(* Logix 5000 project; controller PLC vendor 1 type 14 code 155 rev 32.13; software revision 32.04; part 4 of 5 *)
(* tags used below, declared in another part *)
   Bridge_Timer_Gearing_Delay : TIMER;
   Bridge_Timer_Gearing_Delay_DN_OS : BOOL;
   Bridge_Timer_Gearing_Duration : TIMER;
   Bridge_Timer_Gearing_Duration_DN_OS : BOOL;
   Bypass_Encoder : BOOL;   // HMI ENABLE ENCODER
   Depositor : Depositor_R2b;
   Depositor_Bridge_Up : BOOL;
   Depositor_Spout_Done_OS : BOOL[32];
   Encoder_Conveyor : AXIS_CIP_DRIVE;
   IO : IO_R2a;
   MV_conveyor_stopped : BOOL;
   MV_Encoder_Stop_Value : REAL;
   mv_index_counter : COUNTER;
   NC_NF : NCNF_R2a;   // NC/NF BITSHIFTS
   OS : INT[10];
   Recipe_Setpoints_DINT : DINT[23,20];
   Release_Bridge_Distance : REAL[10];
   Release_MAG_Distance : REAL[10];
   Releases_Dive : BOOL;
   Sequencer_Auto : Sequencer_R2a;
   Sequencer_Home : Sequencer_R2a;
   Servo_Bridge_Shift : AXIS_CIP_DRIVE;
   Servo_MC_Bridge_Shift : Axis_MC_R3b;
   System : System_R2e;
   TEST_COUNTER : COUNTER;
   TEST_COUNTER_2 : COUNTER;
   Timers : TIMER[20];   // x
(* MainProgram, continued *)

ROUTINE File_100_Servo_Bridge   (* ladder *)
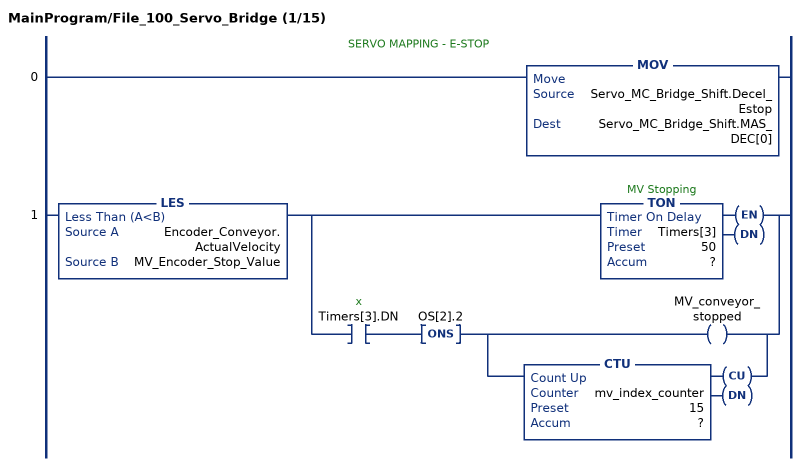
   // SERVO MAPPING - E-STOP
   0: MOV(Servo_MC_Bridge_Shift.Decel_Estop,Servo_MC_Bridge_Shift.MAS_DEC[0]);
   1: LES(Encoder_Conveyor.ActualVelocity,MV_Encoder_Stop_Value)[TON(Timers[3],?,?) ,XIC(Timers[3].DN) ONS(OS[2].2) [OTE(MV_conveyor_stopped) ,CTU(mv_index_counter,?,?) ] ];
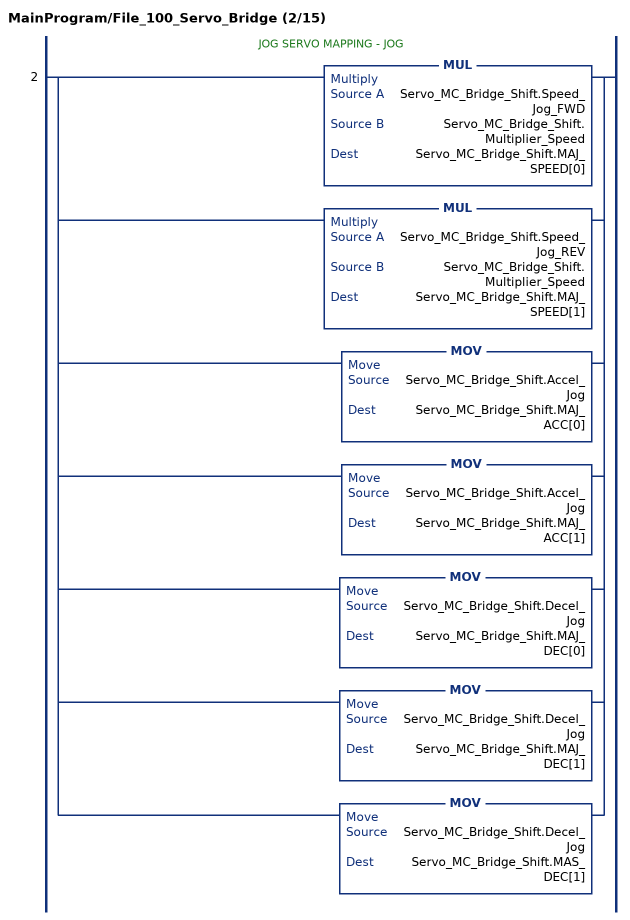
   // JOG SERVO MAPPING - JOG
   2: [MUL(Servo_MC_Bridge_Shift.Speed_Jog_FWD,Servo_MC_Bridge_Shift.Multiplier_Speed,Servo_MC_Bridge_Shift.MAJ_SPEED[0]) ,MUL(Servo_MC_Bridge_Shift.Speed_Jog_REV,Servo_MC_Bridge_Shift.Multiplier_Speed,Servo_MC_Bridge_Shift.MAJ_SPEED[1]) ,MOV(Servo_MC_Bridge_Shift.Accel_Jog,Servo_MC_Bridge_Shift.MAJ_ACC[0]) ,MOV(Servo_MC_Bridge_Shift.Accel_Jog,Servo_MC_Bridge_Shift.MAJ_ACC[1]) ,MOV(Servo_MC_Bridge_Shift.Decel_Jog,Servo_MC_Bridge_Shift.MAJ_DEC[0]) ,MOV(Servo_MC_Bridge_Shift.Decel_Jog,Servo_MC_Bridge_Shift.MAJ_DEC[1]) ,MOV(Servo_MC_Bridge_Shift.Decel_Jog,Servo_MC_Bridge_Shift.MAS_DEC[1]) ];
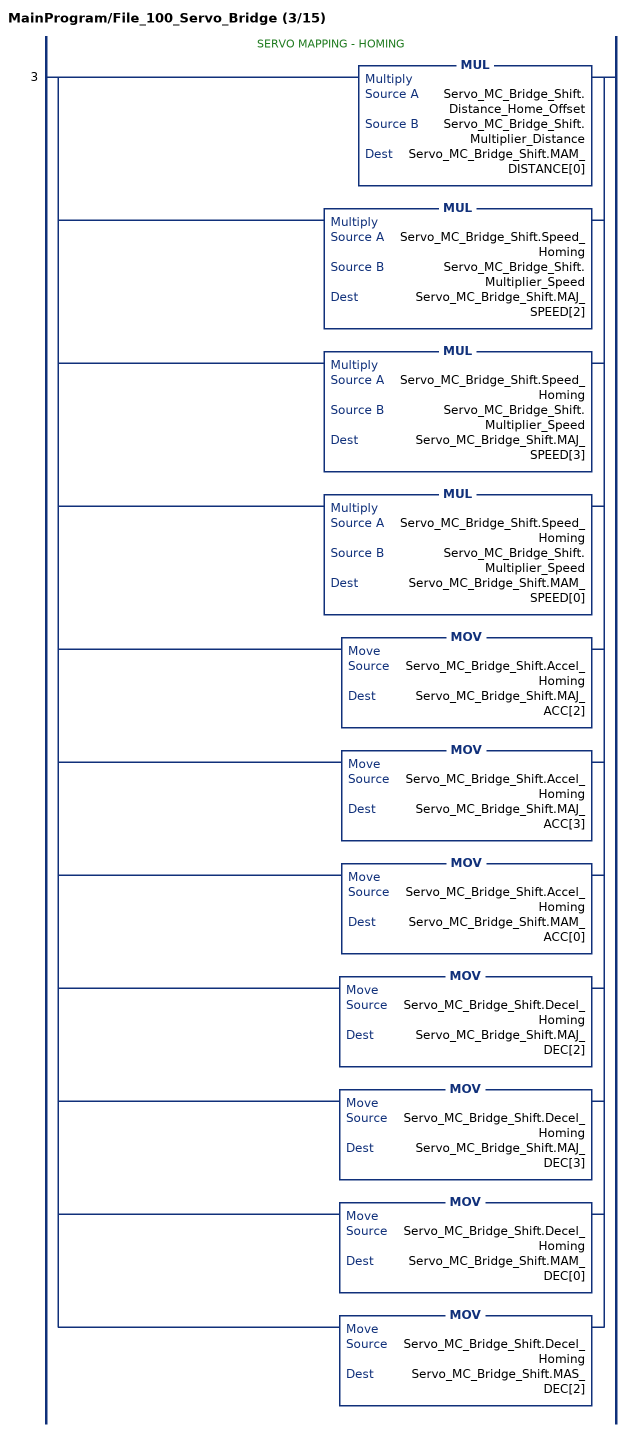
   // SERVO MAPPING - HOMING
   3: [MUL(Servo_MC_Bridge_Shift.Distance_Home_Offset,Servo_MC_Bridge_Shift.Multiplier_Distance,Servo_MC_Bridge_Shift.MAM_DISTANCE[0]) ,MUL(Servo_MC_Bridge_Shift.Speed_Homing,Servo_MC_Bridge_Shift.Multiplier_Speed,Servo_MC_Bridge_Shift.MAJ_SPEED[2]) ,MUL(Servo_MC_Bridge_Shift.Speed_Homing,Servo_MC_Bridge_Shift.Multiplier_Speed,Servo_MC_Bridge_Shift.MAJ_SPEED[3]) ,MUL(Servo_MC_Bridge_Shift.Speed_Homing,Servo_MC_Bridge_Shift.Multiplier_Speed,Servo_MC_Bridge_Shift.MAM_SPEED[0]) ,MOV(Servo_MC_Bridge_Shift.Accel_Homing,Servo_MC_Bridge_Shift.MAJ_ACC[2]) ,MOV(Servo_MC_Bridge_Shift.Accel_Homing,Servo_MC_Bridge_Shift.MAJ_ACC[3]) ,MOV(Servo_MC_Bridge_Shift.Accel_Homing,Servo_MC_Bridge_Shift.MAM_ACC[0]) ,MOV(Servo_MC_Bridge_Shift.Decel_Homing,Servo_MC_Bridge_Shift.MAJ_DEC[2]) ,MOV(Servo_MC_Bridge_Shift.Decel_Homing,Servo_MC_Bridge_Shift.MAJ_DEC[3]) ,MOV(Servo_MC_Bridge_Shift.Decel_Homing,Servo_MC_Bridge_Shift.MAM_DEC[0]) ,MOV(Servo_MC_Bridge_Shift.Decel_Homing,Servo_MC_Bridge_Shift.MAS_DEC[2]) ];
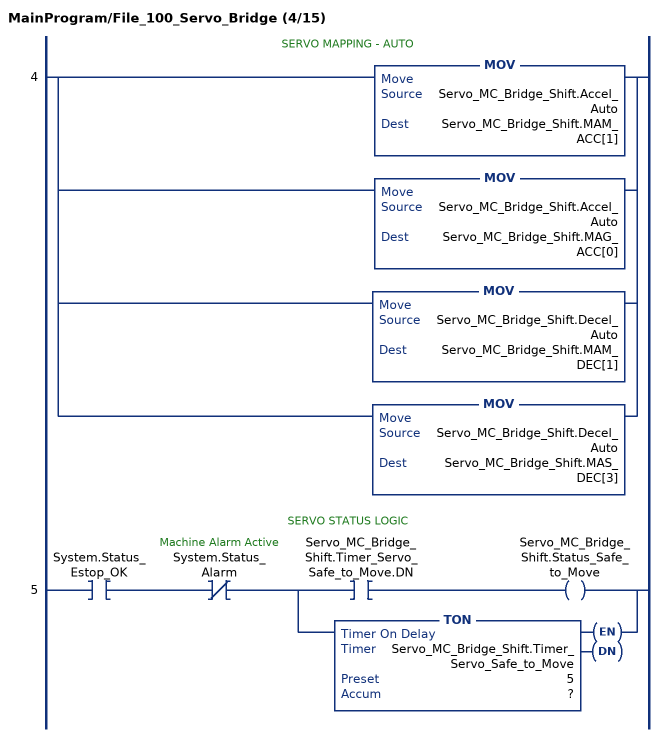
   // SERVO MAPPING - AUTO
   4: [MOV(Servo_MC_Bridge_Shift.Accel_Auto,Servo_MC_Bridge_Shift.MAM_ACC[1]) ,MOV(Servo_MC_Bridge_Shift.Accel_Auto,Servo_MC_Bridge_Shift.MAG_ACC[0]) ,MOV(Servo_MC_Bridge_Shift.Decel_Auto,Servo_MC_Bridge_Shift.MAM_DEC[1]) ,MOV(Servo_MC_Bridge_Shift.Decel_Auto,Servo_MC_Bridge_Shift.MAS_DEC[3]) ];
   // SERVO STATUS LOGIC
   5: XIC(System.Status_Estop_OK)XIO(System.Status_Alarm)[XIC(Servo_MC_Bridge_Shift.Timer_Servo_Safe_to_Move.DN) OTE(Servo_MC_Bridge_Shift.Status_Safe_to_Move) ,TON(Servo_MC_Bridge_Shift.Timer_Servo_Safe_to_Move,?,?) ];
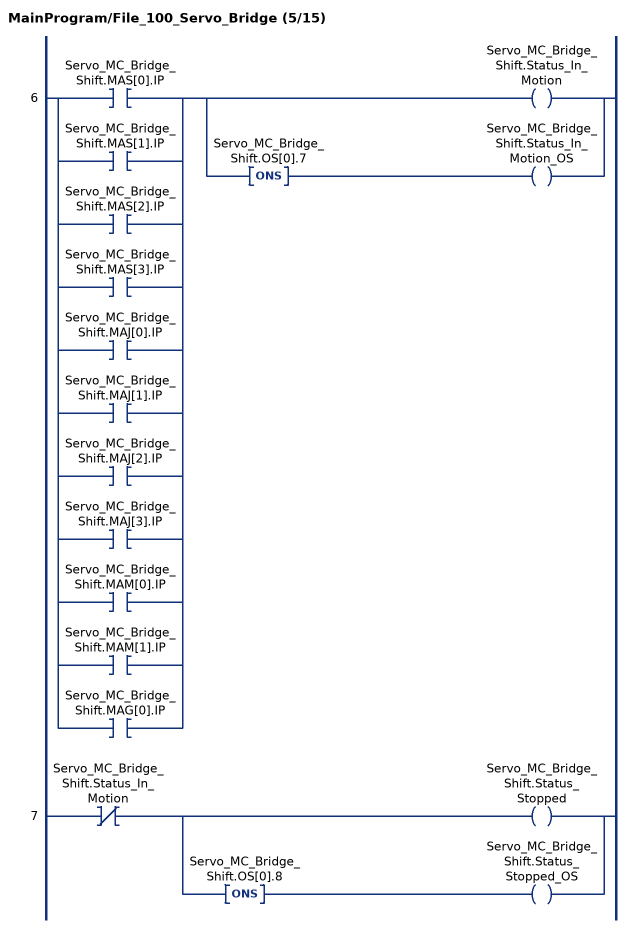
   6: [XIC(Servo_MC_Bridge_Shift.MAS[0].IP) ,XIC(Servo_MC_Bridge_Shift.MAS[1].IP) ,XIC(Servo_MC_Bridge_Shift.MAS[2].IP) ,XIC(Servo_MC_Bridge_Shift.MAS[3].IP) ,XIC(Servo_MC_Bridge_Shift.MAJ[0].IP) ,XIC(Servo_MC_Bridge_Shift.MAJ[1].IP) ,XIC(Servo_MC_Bridge_Shift.MAJ[2].IP) ,XIC(Servo_MC_Bridge_Shift.MAJ[3].IP) ,XIC(Servo_MC_Bridge_Shift.MAM[0].IP) ,XIC(Servo_MC_Bridge_Shift.MAM[1].IP) ,XIC(Servo_MC_Bridge_Shift.MAG[0].IP) ][OTE(Servo_MC_Bridge_Shift.Status_In_Motion) ,ONS(Servo_MC_Bridge_Shift.OS[0].7) OTE(Servo_MC_Bridge_Shift.Status_In_Motion_OS) ];
   7: XIO(Servo_MC_Bridge_Shift.Status_In_Motion)[OTE(Servo_MC_Bridge_Shift.Status_Stopped) ,ONS(Servo_MC_Bridge_Shift.OS[0].8) OTE(Servo_MC_Bridge_Shift.Status_Stopped_OS) ];
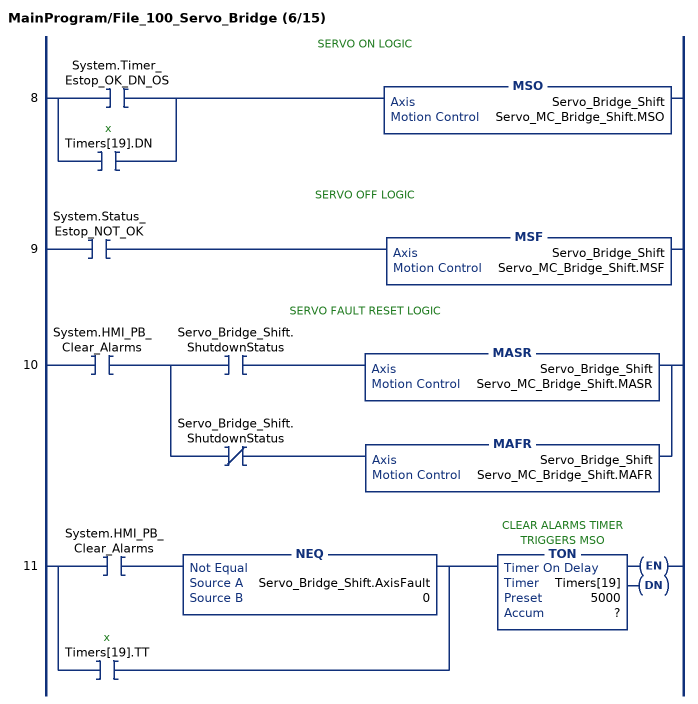
   // SERVO ON LOGIC
   8: [XIC(System.Timer_Estop_OK_DN_OS) ,XIC(Timers[19].DN) ]MSO(Servo_Bridge_Shift,Servo_MC_Bridge_Shift.MSO);
   // SERVO OFF LOGIC
   9: XIC(System.Status_Estop_NOT_OK)MSF(Servo_Bridge_Shift,Servo_MC_Bridge_Shift.MSF);
   // SERVO FAULT RESET LOGIC
   10: XIC(System.HMI_PB_Clear_Alarms)[XIC(Servo_Bridge_Shift.ShutdownStatus) MASR(Servo_Bridge_Shift,Servo_MC_Bridge_Shift.MASR) ,XIO(Servo_Bridge_Shift.ShutdownStatus) MAFR(Servo_Bridge_Shift,Servo_MC_Bridge_Shift.MAFR) ];
   11: [XIC(System.HMI_PB_Clear_Alarms) NEQ(Servo_Bridge_Shift.AxisFault,0) ,XIC(Timers[19].TT) ]TON(Timers[19],?,?);
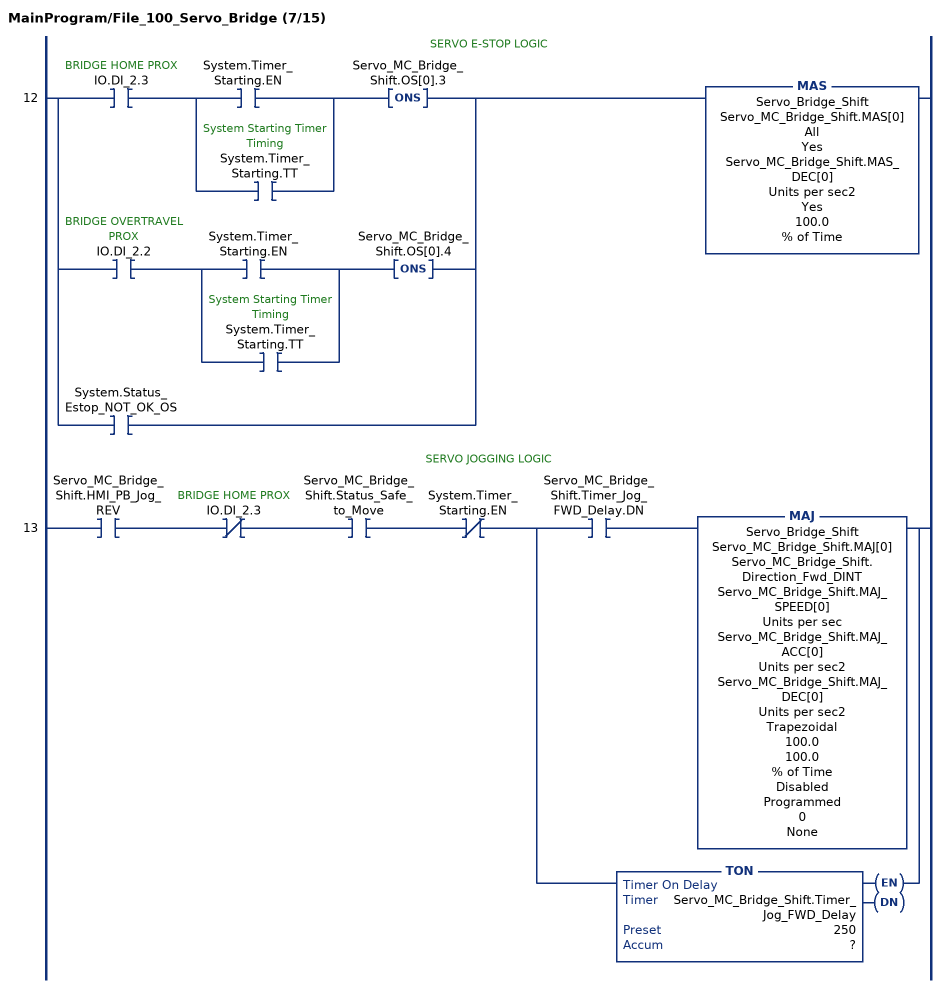
   // SERVO E-STOP LOGIC
   12: [XIC(IO.DI_2.3) [XIC(System.Timer_Starting.EN) ,XIC(System.Timer_Starting.TT) ] ONS(Servo_MC_Bridge_Shift.OS[0].3) ,XIC(IO.DI_2.2) [XIC(System.Timer_Starting.EN) ,XIC(System.Timer_Starting.TT) ] ONS(Servo_MC_Bridge_Shift.OS[0].4) ,XIC(System.Status_Estop_NOT_OK_OS) ]MAS(Servo_Bridge_Shift,Servo_MC_Bridge_Shift.MAS[0],All,Yes,Servo_MC_Bridge_Shift.MAS_DEC[0],Units per sec2,Yes,100.0,% of Time);
   // SERVO JOGGING LOGIC
   13: XIC(Servo_MC_Bridge_Shift.HMI_PB_Jog_REV)XIO(IO.DI_2.3)XIC(Servo_MC_Bridge_Shift.Status_Safe_to_Move)XIO(System.Timer_Starting.EN)[XIC(Servo_MC_Bridge_Shift.Timer_Jog_FWD_Delay.DN) MAJ(Servo_Bridge_Shift,Servo_MC_Bridge_Shift.MAJ[0],Servo_MC_Bridge_Shift.Direction_Fwd_DINT,Servo_MC_Bridge_Shift.MAJ_SPEED[0],Units per sec,Servo_MC_Bridge_Shift.MAJ_ACC[0],Units per sec2,Servo_MC_Bridge_Shift.MAJ_DEC[0],Units per sec2,Trapezoidal,100.0,100.0,% of Time,Disabled,Programmed,0,None) ,TON(Servo_MC_Bridge_Shift.Timer_Jog_FWD_Delay,?,?) ];
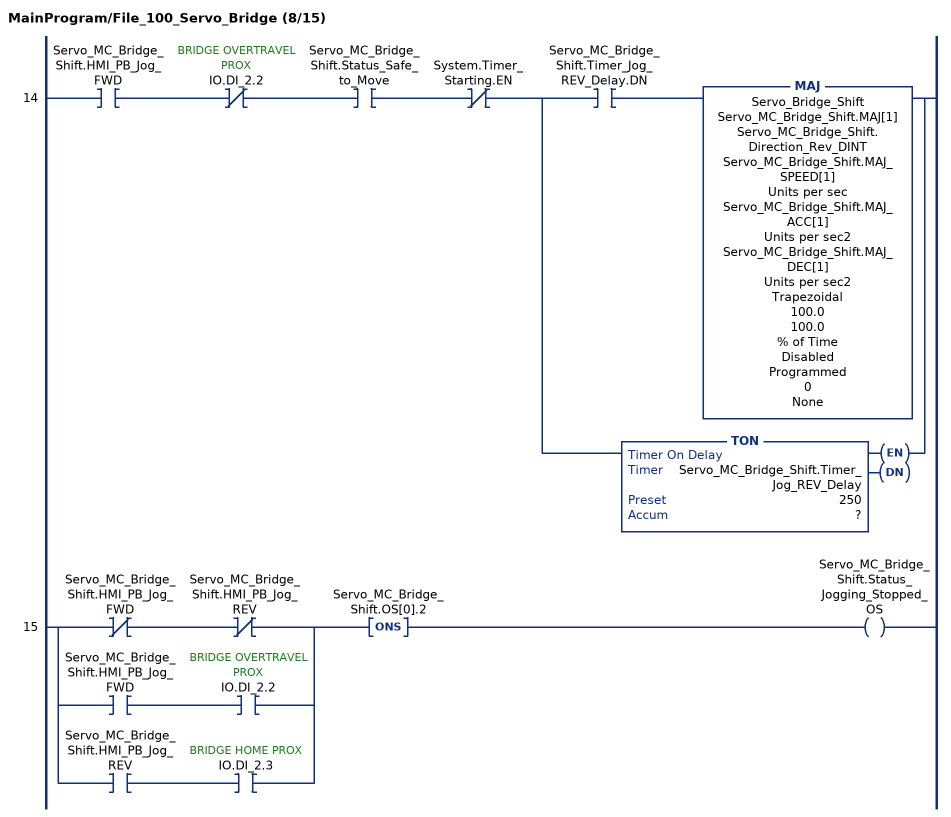
   14: XIC(Servo_MC_Bridge_Shift.HMI_PB_Jog_FWD)XIO(IO.DI_2.2)XIC(Servo_MC_Bridge_Shift.Status_Safe_to_Move)XIO(System.Timer_Starting.EN)[XIC(Servo_MC_Bridge_Shift.Timer_Jog_REV_Delay.DN) MAJ(Servo_Bridge_Shift,Servo_MC_Bridge_Shift.MAJ[1],Servo_MC_Bridge_Shift.Direction_Rev_DINT,Servo_MC_Bridge_Shift.MAJ_SPEED[1],Units per sec,Servo_MC_Bridge_Shift.MAJ_ACC[1],Units per sec2,Servo_MC_Bridge_Shift.MAJ_DEC[1],Units per sec2,Trapezoidal,100.0,100.0,% of Time,Disabled,Programmed,0,None) ,TON(Servo_MC_Bridge_Shift.Timer_Jog_REV_Delay,?,?) ];
   15: [XIO(Servo_MC_Bridge_Shift.HMI_PB_Jog_FWD) XIO(Servo_MC_Bridge_Shift.HMI_PB_Jog_REV) ,XIC(Servo_MC_Bridge_Shift.HMI_PB_Jog_FWD) XIC(IO.DI_2.2) ,XIC(Servo_MC_Bridge_Shift.HMI_PB_Jog_REV) XIC(IO.DI_2.3) ]ONS(Servo_MC_Bridge_Shift.OS[0].2)OTE(Servo_MC_Bridge_Shift.Status_Jogging_Stopped_OS);
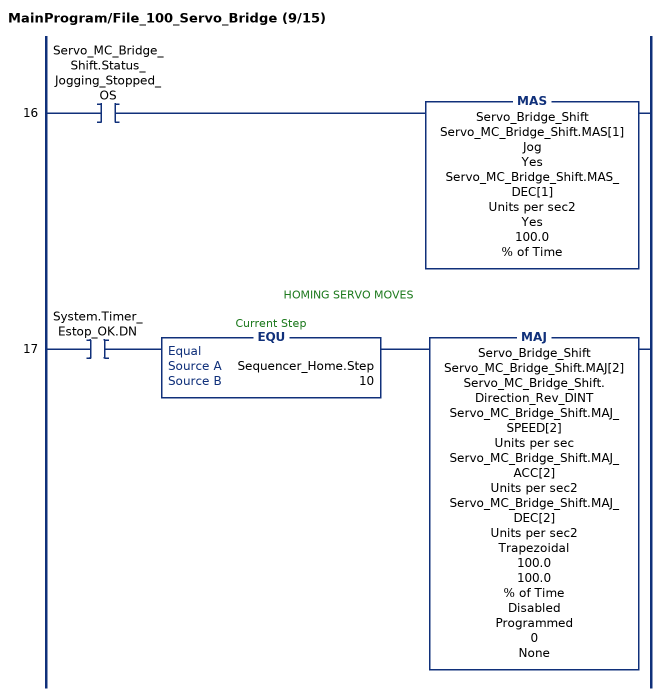
   16: XIC(Servo_MC_Bridge_Shift.Status_Jogging_Stopped_OS)MAS(Servo_Bridge_Shift,Servo_MC_Bridge_Shift.MAS[1],Jog,Yes,Servo_MC_Bridge_Shift.MAS_DEC[1],Units per sec2,Yes,100.0,% of Time);
   // HOMING SERVO MOVES
   17: XIC(System.Timer_Estop_OK.DN)EQU(Sequencer_Home.Step,10)MAJ(Servo_Bridge_Shift,Servo_MC_Bridge_Shift.MAJ[2],Servo_MC_Bridge_Shift.Direction_Rev_DINT,Servo_MC_Bridge_Shift.MAJ_SPEED[2],Units per sec,Servo_MC_Bridge_Shift.MAJ_ACC[2],Units per sec2,Servo_MC_Bridge_Shift.MAJ_DEC[2],Units per sec2,Trapezoidal,100.0,100.0,% of Time,Disabled,Programmed,0,None);
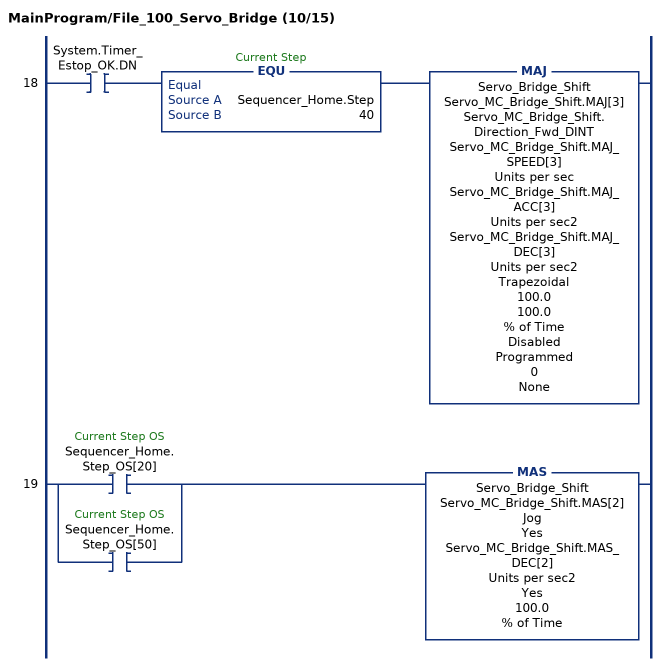
   18: XIC(System.Timer_Estop_OK.DN)EQU(Sequencer_Home.Step,40)MAJ(Servo_Bridge_Shift,Servo_MC_Bridge_Shift.MAJ[3],Servo_MC_Bridge_Shift.Direction_Fwd_DINT,Servo_MC_Bridge_Shift.MAJ_SPEED[3],Units per sec,Servo_MC_Bridge_Shift.MAJ_ACC[3],Units per sec2,Servo_MC_Bridge_Shift.MAJ_DEC[3],Units per sec2,Trapezoidal,100.0,100.0,% of Time,Disabled,Programmed,0,None);
   19: [XIC(Sequencer_Home.Step_OS[20]) ,XIC(Sequencer_Home.Step_OS[50]) ]MAS(Servo_Bridge_Shift,Servo_MC_Bridge_Shift.MAS[2],Jog,Yes,Servo_MC_Bridge_Shift.MAS_DEC[2],Units per sec2,Yes,100.0,% of Time);
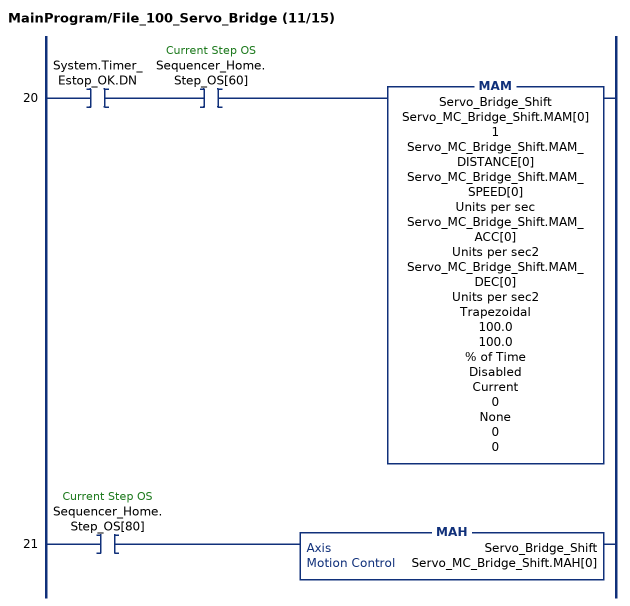
   20: XIC(System.Timer_Estop_OK.DN)XIC(Sequencer_Home.Step_OS[60])MAM(Servo_Bridge_Shift,Servo_MC_Bridge_Shift.MAM[0],1,Servo_MC_Bridge_Shift.MAM_DISTANCE[0],Servo_MC_Bridge_Shift.MAM_SPEED[0],Units per sec,Servo_MC_Bridge_Shift.MAM_ACC[0],Units per sec2,Servo_MC_Bridge_Shift.MAM_DEC[0],Units per sec2,Trapezoidal,100.0,100.0,% of Time,Disabled,Current,0,None,0,0);
   21: XIC(Sequencer_Home.Step_OS[80])MAH(Servo_Bridge_Shift,Servo_MC_Bridge_Shift.MAH[0]);
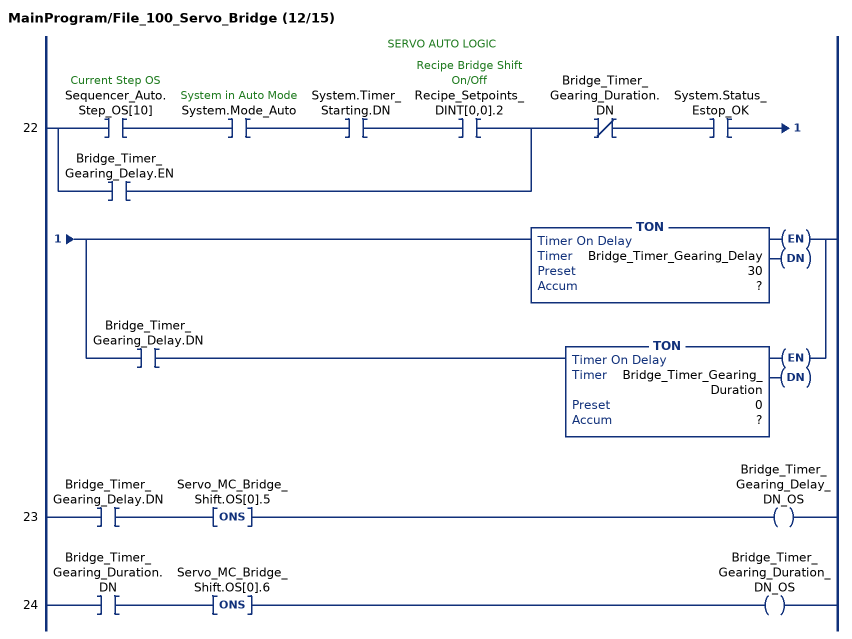
   // SERVO AUTO LOGIC
   22: [XIC(Sequencer_Auto.Step_OS[10]) XIC(System.Mode_Auto) XIC(System.Timer_Starting.DN) XIC(Recipe_Setpoints_DINT[0,0].2) ,XIC(Bridge_Timer_Gearing_Delay.EN) ]XIO(Bridge_Timer_Gearing_Duration.DN)XIC(System.Status_Estop_OK)[TON(Bridge_Timer_Gearing_Delay,?,?) ,XIC(Bridge_Timer_Gearing_Delay.DN) TON(Bridge_Timer_Gearing_Duration,?,?) ];
   23: XIC(Bridge_Timer_Gearing_Delay.DN)ONS(Servo_MC_Bridge_Shift.OS[0].5)OTE(Bridge_Timer_Gearing_Delay_DN_OS);
   24: XIC(Bridge_Timer_Gearing_Duration.DN)ONS(Servo_MC_Bridge_Shift.OS[0].6)OTE(Bridge_Timer_Gearing_Duration_DN_OS);
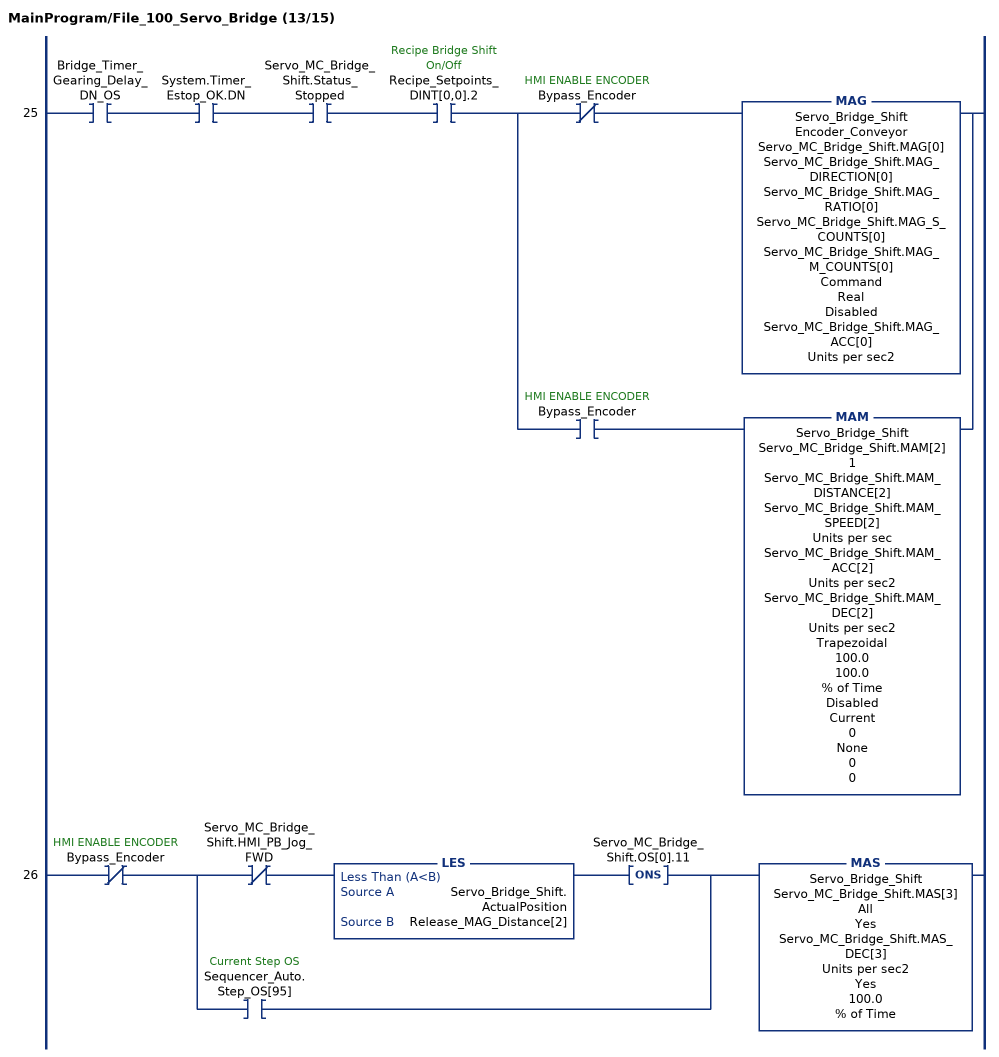
   25: XIC(Bridge_Timer_Gearing_Delay_DN_OS)XIC(System.Timer_Estop_OK.DN)XIC(Servo_MC_Bridge_Shift.Status_Stopped)XIC(Recipe_Setpoints_DINT[0,0].2)[XIO(Bypass_Encoder) MAG(Servo_Bridge_Shift,Encoder_Conveyor,Servo_MC_Bridge_Shift.MAG[0],Servo_MC_Bridge_Shift.MAG_DIRECTION[0],Servo_MC_Bridge_Shift.MAG_RATIO[0],Servo_MC_Bridge_Shift.MAG_S_COUNTS[0],Servo_MC_Bridge_Shift.MAG_M_COUNTS[0],Command,Real,Disabled,Servo_MC_Bridge_Shift.MAG_ACC[0],Units per sec2) ,XIC(Bypass_Encoder) MAM(Servo_Bridge_Shift,Servo_MC_Bridge_Shift.MAM[2],1,Servo_MC_Bridge_Shift.MAM_DISTANCE[2],Servo_MC_Bridge_Shift.MAM_SPEED[2],Units per sec,Servo_MC_Bridge_Shift.MAM_ACC[2],Units per sec2,Servo_MC_Bridge_Shift.MAM_DEC[2],Units per sec2,Trapezoidal,100.0,100.0,% of Time,Disabled,Current,0,None,0,0) ];
   26: XIO(Bypass_Encoder)[XIO(Servo_MC_Bridge_Shift.HMI_PB_Jog_FWD) LES(Servo_Bridge_Shift.ActualPosition,Release_MAG_Distance[2]) ONS(Servo_MC_Bridge_Shift.OS[0].11) ,XIC(Sequencer_Auto.Step_OS[95]) ]MAS(Servo_Bridge_Shift,Servo_MC_Bridge_Shift.MAS[3],All,Yes,Servo_MC_Bridge_Shift.MAS_DEC[3],Units per sec2,Yes,100.0,% of Time);
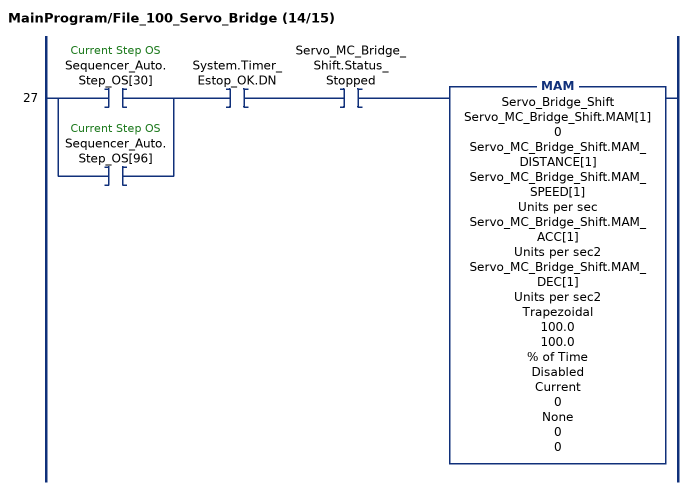
   27: [XIC(Sequencer_Auto.Step_OS[30]) ,XIC(Sequencer_Auto.Step_OS[96]) ]XIC(System.Timer_Estop_OK.DN)XIC(Servo_MC_Bridge_Shift.Status_Stopped)MAM(Servo_Bridge_Shift,Servo_MC_Bridge_Shift.MAM[1],0,Servo_MC_Bridge_Shift.MAM_DISTANCE[1],Servo_MC_Bridge_Shift.MAM_SPEED[1],Units per sec,Servo_MC_Bridge_Shift.MAM_ACC[1],Units per sec2,Servo_MC_Bridge_Shift.MAM_DEC[1],Units per sec2,Trapezoidal,100.0,100.0,% of Time,Disabled,Current,0,None,0,0);
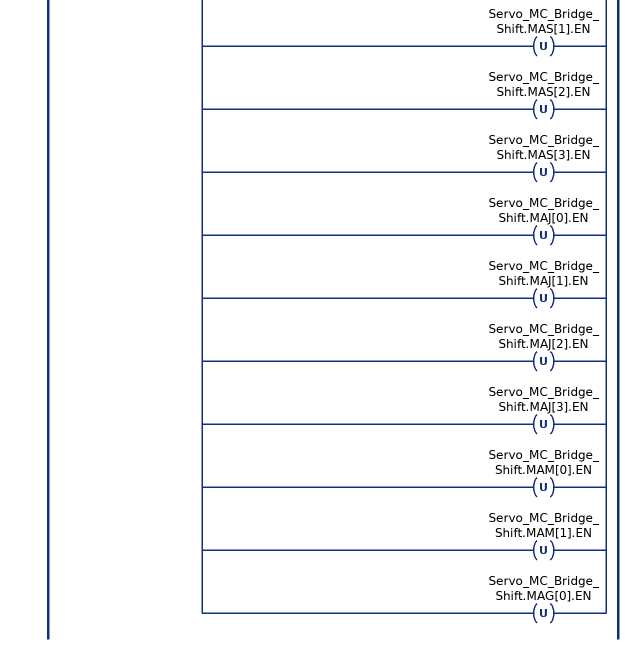
   // MOTION INSTRUCTIONS UNLATCH LOGIC
   28: [XIC(System.Timer_Estop_OK_DN_OS) ,XIC(System.HMI_PB_Clear_Alarms) ,XIC(System.Timer_Starting_TT_OS) ][OTU(Servo_MC_Bridge_Shift.MSO.ER) ,OTU(Servo_MC_Bridge_Shift.MSF.ER) ,OTU(Servo_MC_Bridge_Shift.MAS[0].ER) ,OTU(Servo_MC_Bridge_Shift.MAS[1].ER) ,OTU(Servo_MC_Bridge_Shift.MAS[2].ER) ,OTU(Servo_MC_Bridge_Shift.MAS[3].ER) ,OTU(Servo_MC_Bridge_Shift.MAJ[0].ER) ,OTU(Servo_MC_Bridge_Shift.MAJ[1].ER) ,OTU(Servo_MC_Bridge_Shift.MAJ[2].ER) ,OTU(Servo_MC_Bridge_Shift.MAJ[3].ER) ,OTU(Servo_MC_Bridge_Shift.MAM[0].ER) ,OTU(Servo_MC_Bridge_Shift.MAM[1].ER) ,OTU(Servo_MC_Bridge_Shift.MAG[0].ER) ,OTU(Servo_MC_Bridge_Shift.MSO.EN) ,OTU(Servo_MC_Bridge_Shift.MSF.EN) ,OTU(Servo_MC_Bridge_Shift.MAS[0].EN) ,OTU(Servo_MC_Bridge_Shift.MAS[1].EN) ,OTU(Servo_MC_Bridge_Shift.MAS[2].EN) ,OTU(Servo_MC_Bridge_Shift.MAS[3].EN) ,OTU(Servo_MC_Bridge_Shift.MAJ[0].EN) ,OTU(Servo_MC_Bridge_Shift.MAJ[1].EN) ,OTU(Servo_MC_Bridge_Shift.MAJ[2].EN) ,OTU(Servo_MC_Bridge_Shift.MAJ[3].EN) ,OTU(Servo_MC_Bridge_Shift.MAM[0].EN) ,OTU(Servo_MC_Bridge_Shift.MAM[1].EN) ,OTU(Servo_MC_Bridge_Shift.MAG[0].EN) ];
END_ROUTINE

ROUTINE File_200_Depositor   (* ladder *)
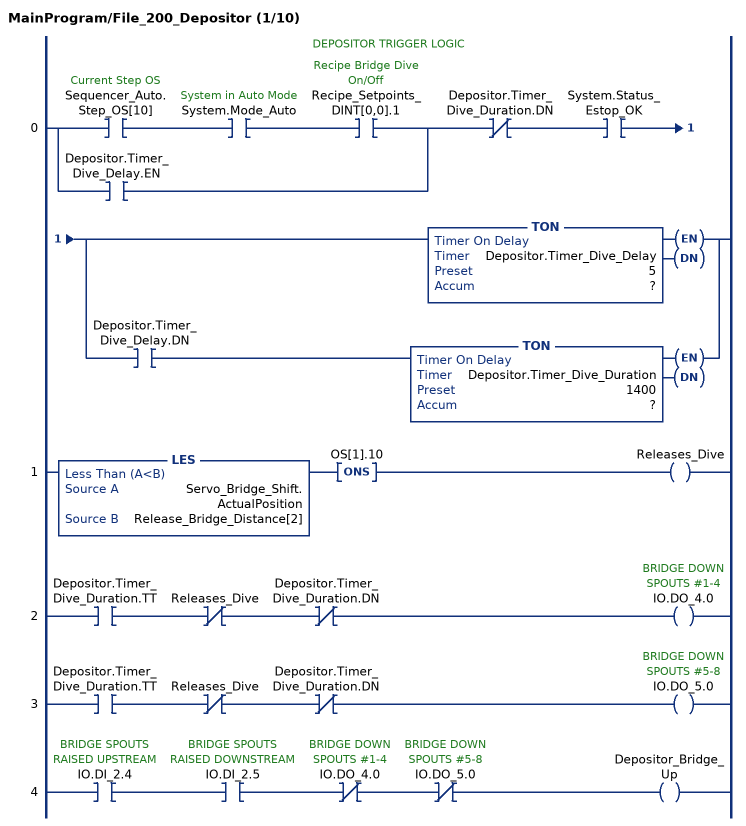
   // DEPOSITOR TRIGGER LOGIC
   0: [XIC(Sequencer_Auto.Step_OS[10]) XIC(System.Mode_Auto) XIC(Recipe_Setpoints_DINT[0,0].1) ,XIC(Depositor.Timer_Dive_Delay.EN) ]XIO(Depositor.Timer_Dive_Duration.DN)XIC(System.Status_Estop_OK)[TON(Depositor.Timer_Dive_Delay,?,?) ,XIC(Depositor.Timer_Dive_Delay.DN) TON(Depositor.Timer_Dive_Duration,?,?) ];
   1: LES(Servo_Bridge_Shift.ActualPosition,Release_Bridge_Distance[2])ONS(OS[1].10)OTE(Releases_Dive);
   2: XIC(Depositor.Timer_Dive_Duration.TT)XIO(Releases_Dive)XIO(Depositor.Timer_Dive_Duration.DN)OTE(IO.DO_4.0);
   3: XIC(Depositor.Timer_Dive_Duration.TT)XIO(Releases_Dive)XIO(Depositor.Timer_Dive_Duration.DN)OTE(IO.DO_5.0);
   4: XIC(IO.DI_2.4)XIC(IO.DI_2.5)XIO(IO.DO_4.0)XIO(IO.DO_5.0)OTE(Depositor_Bridge_Up);
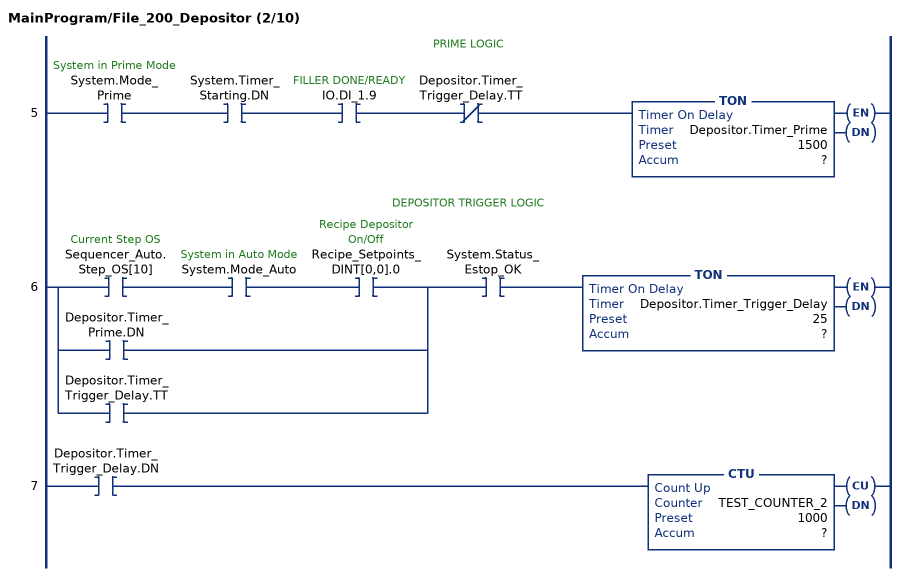
   // PRIME LOGIC
   5: XIC(System.Mode_Prime)XIC(System.Timer_Starting.DN)XIC(IO.DI_1.9)XIO(Depositor.Timer_Trigger_Delay.TT)TON(Depositor.Timer_Prime,?,?);
   // DEPOSITOR TRIGGER LOGIC
   6: [XIC(Sequencer_Auto.Step_OS[10]) XIC(System.Mode_Auto) XIC(Recipe_Setpoints_DINT[0,0].0) ,XIC(Depositor.Timer_Prime.DN) ,XIC(Depositor.Timer_Trigger_Delay.TT) ]XIC(System.Status_Estop_OK)TON(Depositor.Timer_Trigger_Delay,?,?);
   7: XIC(Depositor.Timer_Trigger_Delay.DN)CTU(TEST_COUNTER_2,?,?);
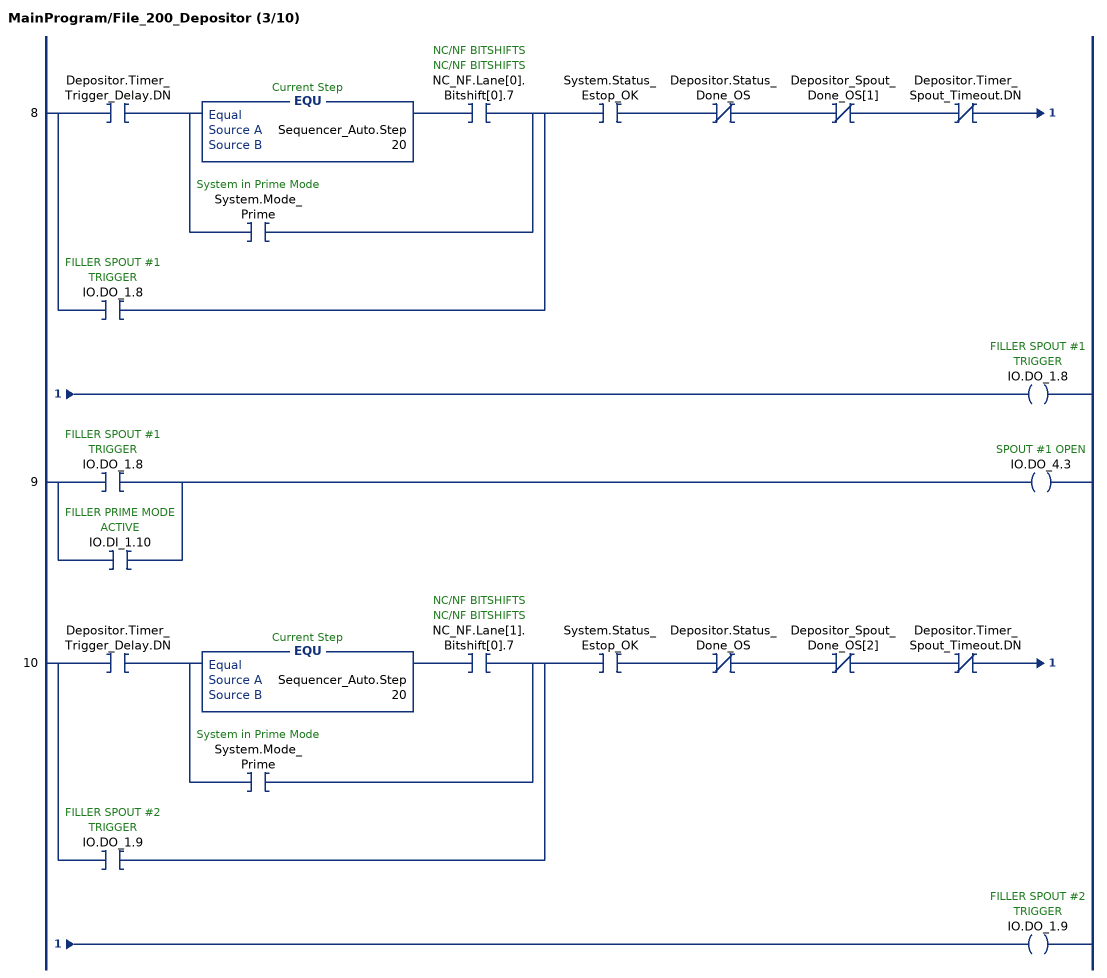
   8: [XIC(Depositor.Timer_Trigger_Delay.DN) [EQU(Sequencer_Auto.Step,20) XIC(NC_NF.Lane[0].Bitshift[0].7) ,XIC(System.Mode_Prime) ] ,XIC(IO.DO_1.8) ]XIC(System.Status_Estop_OK)XIO(Depositor.Status_Done_OS)XIO(Depositor_Spout_Done_OS[1])XIO(Depositor.Timer_Spout_Timeout.DN)OTE(IO.DO_1.8);
   9: [XIC(IO.DO_1.8) ,XIC(IO.DI_1.10) ]OTE(IO.DO_4.3);
   10: [XIC(Depositor.Timer_Trigger_Delay.DN) [EQU(Sequencer_Auto.Step,20) XIC(NC_NF.Lane[1].Bitshift[0].7) ,XIC(System.Mode_Prime) ] ,XIC(IO.DO_1.9) ]XIC(System.Status_Estop_OK)XIO(Depositor.Status_Done_OS)XIO(Depositor_Spout_Done_OS[2])XIO(Depositor.Timer_Spout_Timeout.DN)OTE(IO.DO_1.9);
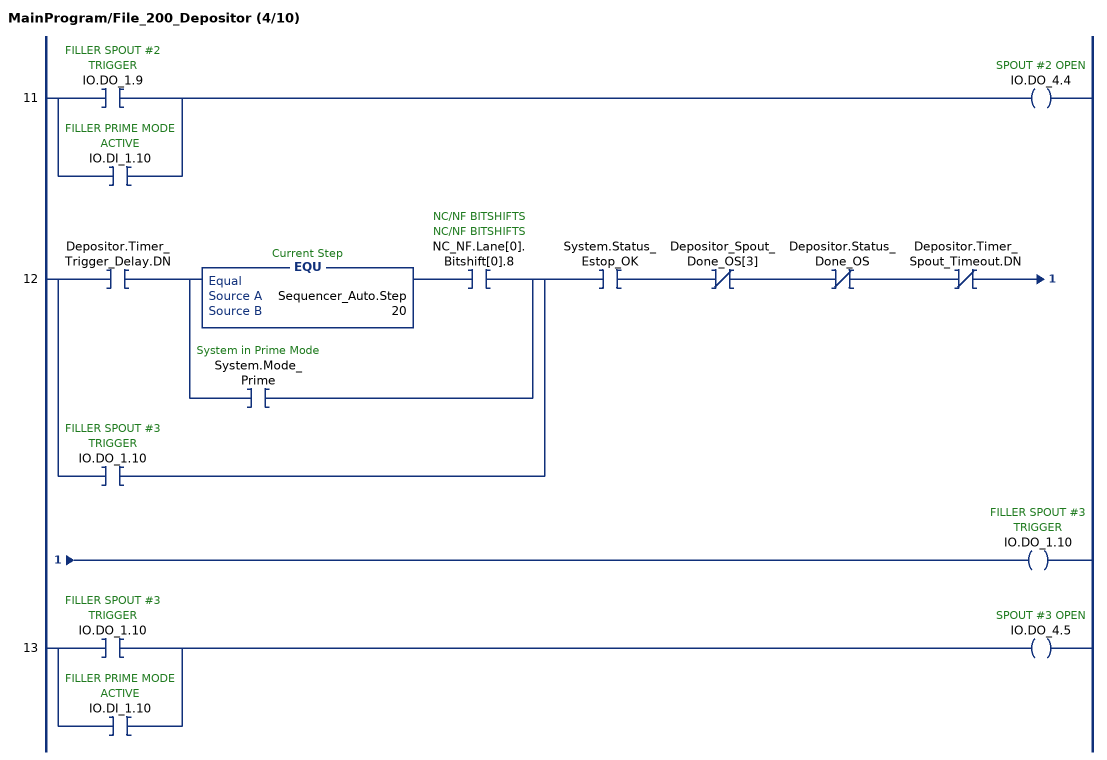
   11: [XIC(IO.DO_1.9) ,XIC(IO.DI_1.10) ]OTE(IO.DO_4.4);
   12: [XIC(Depositor.Timer_Trigger_Delay.DN) [EQU(Sequencer_Auto.Step,20) XIC(NC_NF.Lane[0].Bitshift[0].8) ,XIC(System.Mode_Prime) ] ,XIC(IO.DO_1.10) ]XIC(System.Status_Estop_OK)XIO(Depositor_Spout_Done_OS[3])XIO(Depositor.Status_Done_OS)XIO(Depositor.Timer_Spout_Timeout.DN)OTE(IO.DO_1.10);
   13: [XIC(IO.DO_1.10) ,XIC(IO.DI_1.10) ]OTE(IO.DO_4.5);
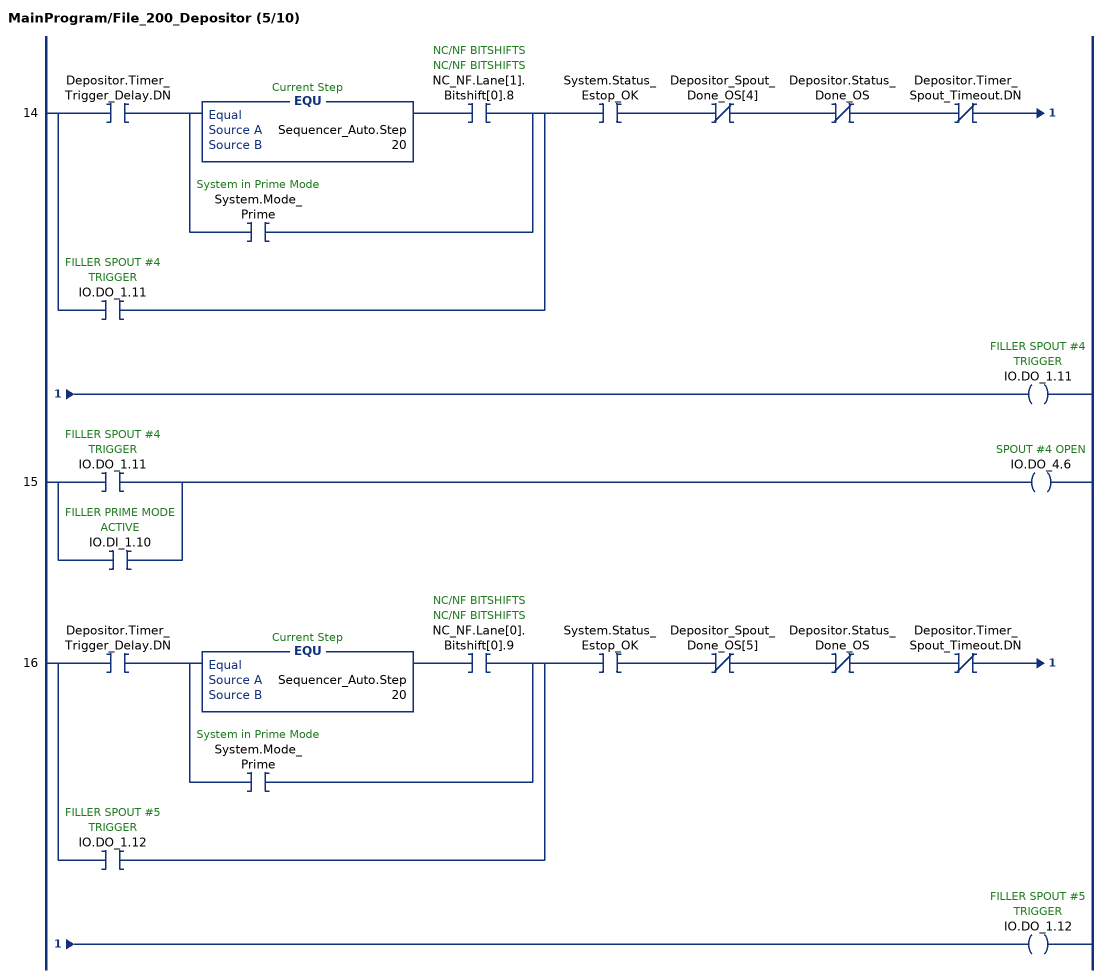
   14: [XIC(Depositor.Timer_Trigger_Delay.DN) [EQU(Sequencer_Auto.Step,20) XIC(NC_NF.Lane[1].Bitshift[0].8) ,XIC(System.Mode_Prime) ] ,XIC(IO.DO_1.11) ]XIC(System.Status_Estop_OK)XIO(Depositor_Spout_Done_OS[4])XIO(Depositor.Status_Done_OS)XIO(Depositor.Timer_Spout_Timeout.DN)OTE(IO.DO_1.11);
   15: [XIC(IO.DO_1.11) ,XIC(IO.DI_1.10) ]OTE(IO.DO_4.6);
   16: [XIC(Depositor.Timer_Trigger_Delay.DN) [EQU(Sequencer_Auto.Step,20) XIC(NC_NF.Lane[0].Bitshift[0].9) ,XIC(System.Mode_Prime) ] ,XIC(IO.DO_1.12) ]XIC(System.Status_Estop_OK)XIO(Depositor_Spout_Done_OS[5])XIO(Depositor.Status_Done_OS)XIO(Depositor.Timer_Spout_Timeout.DN)OTE(IO.DO_1.12);
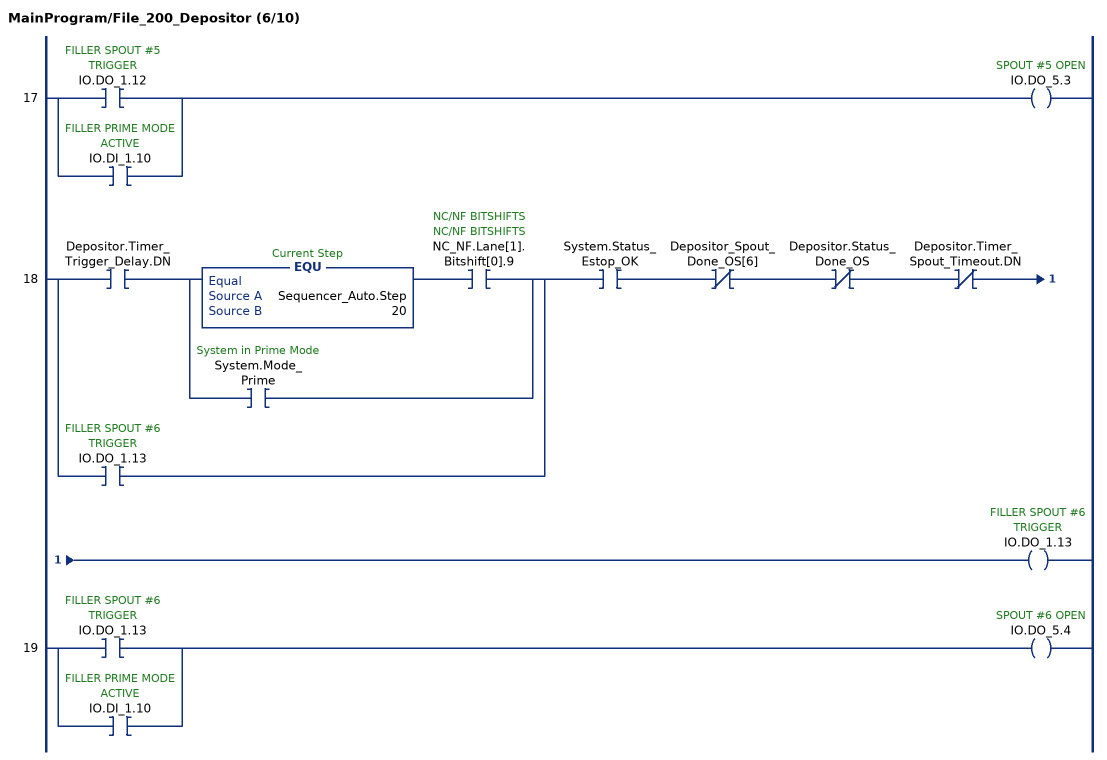
   17: [XIC(IO.DO_1.12) ,XIC(IO.DI_1.10) ]OTE(IO.DO_5.3);
   18: [XIC(Depositor.Timer_Trigger_Delay.DN) [EQU(Sequencer_Auto.Step,20) XIC(NC_NF.Lane[1].Bitshift[0].9) ,XIC(System.Mode_Prime) ] ,XIC(IO.DO_1.13) ]XIC(System.Status_Estop_OK)XIO(Depositor_Spout_Done_OS[6])XIO(Depositor.Status_Done_OS)XIO(Depositor.Timer_Spout_Timeout.DN)OTE(IO.DO_1.13);
   19: [XIC(IO.DO_1.13) ,XIC(IO.DI_1.10) ]OTE(IO.DO_5.4);
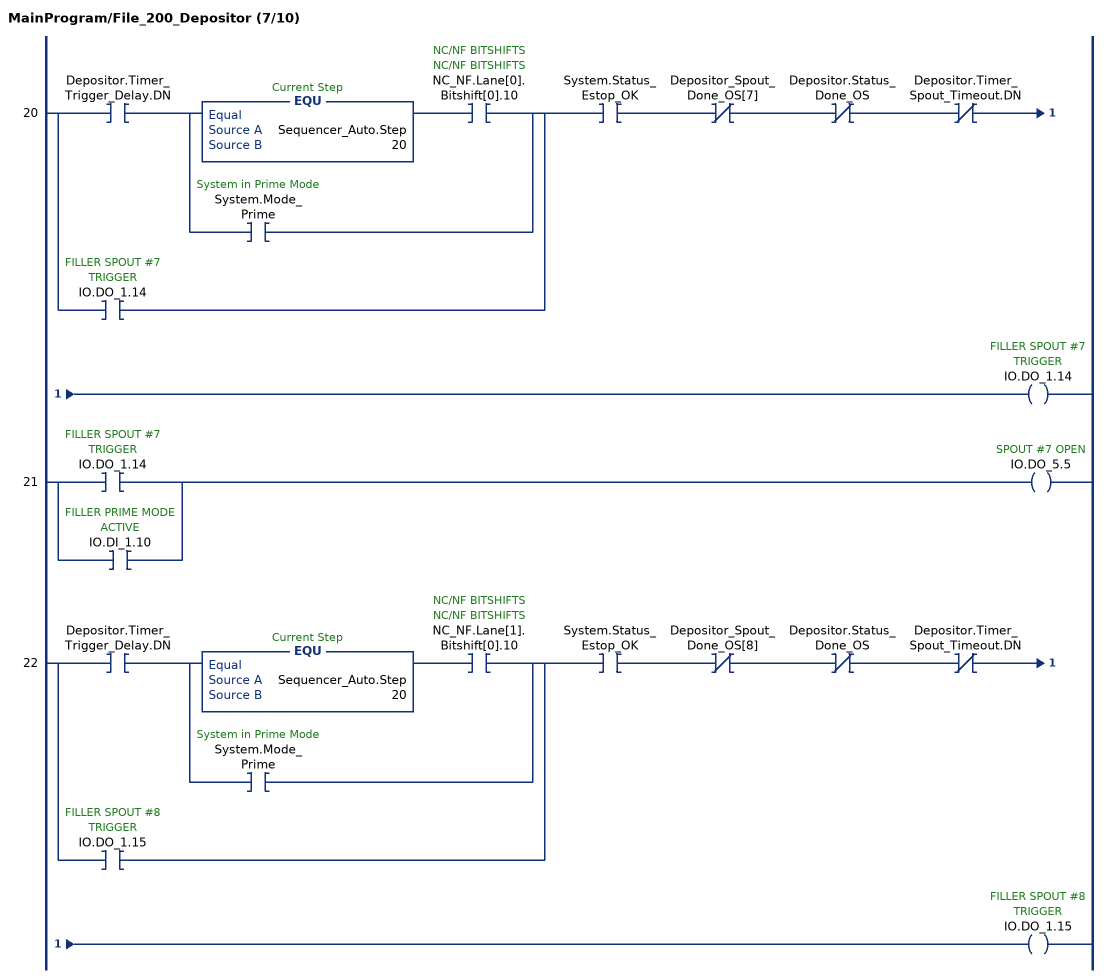
   20: [XIC(Depositor.Timer_Trigger_Delay.DN) [EQU(Sequencer_Auto.Step,20) XIC(NC_NF.Lane[0].Bitshift[0].10) ,XIC(System.Mode_Prime) ] ,XIC(IO.DO_1.14) ]XIC(System.Status_Estop_OK)XIO(Depositor_Spout_Done_OS[7])XIO(Depositor.Status_Done_OS)XIO(Depositor.Timer_Spout_Timeout.DN)OTE(IO.DO_1.14);
   21: [XIC(IO.DO_1.14) ,XIC(IO.DI_1.10) ]OTE(IO.DO_5.5);
   22: [XIC(Depositor.Timer_Trigger_Delay.DN) [EQU(Sequencer_Auto.Step,20) XIC(NC_NF.Lane[1].Bitshift[0].10) ,XIC(System.Mode_Prime) ] ,XIC(IO.DO_1.15) ]XIC(System.Status_Estop_OK)XIO(Depositor_Spout_Done_OS[8])XIO(Depositor.Status_Done_OS)XIO(Depositor.Timer_Spout_Timeout.DN)OTE(IO.DO_1.15);
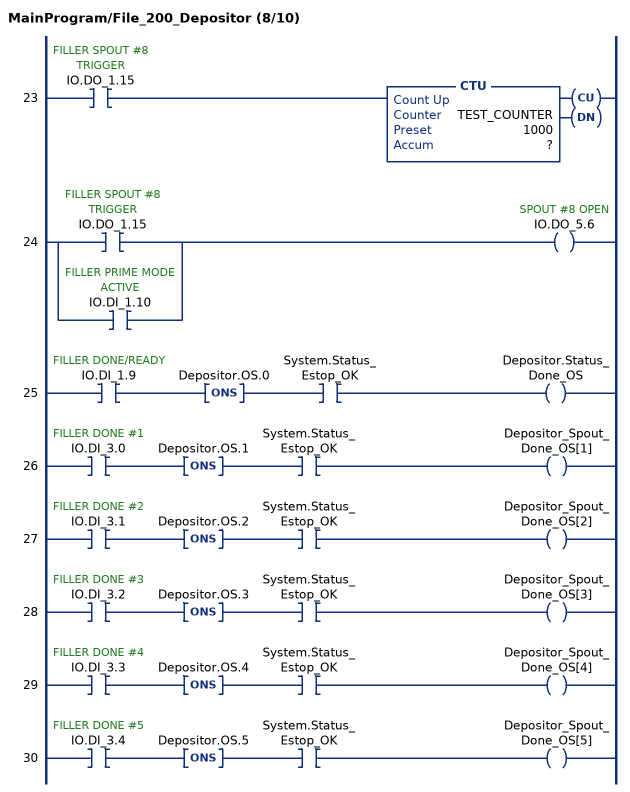
   23: XIC(IO.DO_1.15)CTU(TEST_COUNTER,?,?);
   24: [XIC(IO.DO_1.15) ,XIC(IO.DI_1.10) ]OTE(IO.DO_5.6);
   25: XIC(IO.DI_1.9)ONS(Depositor.OS.0)XIC(System.Status_Estop_OK)OTE(Depositor.Status_Done_OS);
   26: XIC(IO.DI_3.0)ONS(Depositor.OS.1)XIC(System.Status_Estop_OK)OTE(Depositor_Spout_Done_OS[1]);
   27: XIC(IO.DI_3.1)ONS(Depositor.OS.2)XIC(System.Status_Estop_OK)OTE(Depositor_Spout_Done_OS[2]);
   28: XIC(IO.DI_3.2)ONS(Depositor.OS.3)XIC(System.Status_Estop_OK)OTE(Depositor_Spout_Done_OS[3]);
   29: XIC(IO.DI_3.3)ONS(Depositor.OS.4)XIC(System.Status_Estop_OK)OTE(Depositor_Spout_Done_OS[4]);
   30: XIC(IO.DI_3.4)ONS(Depositor.OS.5)XIC(System.Status_Estop_OK)OTE(Depositor_Spout_Done_OS[5]);
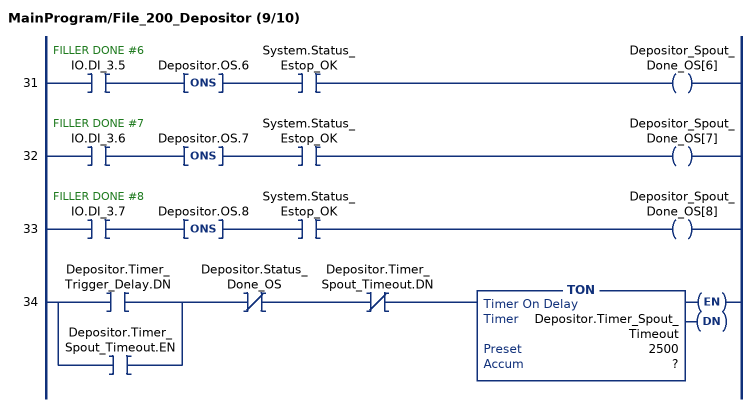
   31: XIC(IO.DI_3.5)ONS(Depositor.OS.6)XIC(System.Status_Estop_OK)OTE(Depositor_Spout_Done_OS[6]);
   32: XIC(IO.DI_3.6)ONS(Depositor.OS.7)XIC(System.Status_Estop_OK)OTE(Depositor_Spout_Done_OS[7]);
   33: XIC(IO.DI_3.7)ONS(Depositor.OS.8)XIC(System.Status_Estop_OK)OTE(Depositor_Spout_Done_OS[8]);
   34: [XIC(Depositor.Timer_Trigger_Delay.DN) ,XIC(Depositor.Timer_Spout_Timeout.EN) ]XIO(Depositor.Status_Done_OS)XIO(Depositor.Timer_Spout_Timeout.DN)TON(Depositor.Timer_Spout_Timeout,?,?);
